Staubli VAL3: exeSE.pgx

program exeSE(dio x_dInput, dio x_dOutput, num x_nLength)
begin

  while true
    x_dOutput=false
    wait(x_dInput==true)
    if !watch(x_dInput==false,x_nLength)
      x_dOutput=true
    endIf
    wait(x_dInput==false)
    x_dOutput=false
  endWhile

end
